FUNCTION_BLOCK FB_DriveInv IMPLEMENTS I_Drive
VAR
	//HMI
	_autoLed			: FB_Led;			//obiekt diody LED stacyjka SCADA - auto
	_supplyLed			: FB_Led;			//obiekt diody LED stacyjka SCADA - zasilanie
	_fwdLed				: FB_Led;			//obiekt diody LED Stacyjka SCADA - kierunek
	_revLed				: FB_LED;			//obiekt diody LED Stacyjka SCADA - kierunek do tyłu
	_stateLed			: FB_LedColorful;	//obiekt etykiety LABEL stacyjka SCADA
	_statusLabel    	: FB_Label;			//obiekt etykiety LABEL sstatus


	// Latch RUN tylko w Drive
    _reqFwd, _reqRev 	: BOOL;
	_fault			 	: BOOL;
	
	// poziomy do styczników
    _cmdFwd, _cmdRev 	: BOOL;
	
	//zezwolenia
	_safetyOk       	: BOOL := TRUE;	// Zawsze TRUE jesli brak przekazników safety
    _permOk	 		 	: BOOL := TRUE;    // „zawsze TRUE”, jeśli brak per-permitu
	
		
	// instancje styczników – referencje wiązane w FB_init
    Fwd					: FB_Contactor( en := _cmdFwd);
    Rev 				: FB_Contactor( en := _cmdRev);
	
	//stan napędu
	_termFuseOk		 	: FB_TermFuse;		//obiekt wylacznika silnikowego fizyczne szafa sterownicza
	_isRunning		 	: BOOL; 
	_isRunningRev 	 	: BOOL;
	
	//czas pracy
	_fbWorkTimeCounter	: FB_WorkTimeCounter; //obiekt do zarzadzania czasem pracy napędu
	_stWorkTime			: ST_WorkTime;		 //struktura przechowywania czasu pracy
	_wtEnable			: BOOL;				//uruchamia licznik czasu pracy
	
	//nastawa i aktualna czestotliwość w HZ pracy
	_rSetHz 			: REAL;   // bufor nastawy (ostatnio zadane)
    _rActHz				: REAL;   // ostatni odczyt z falownika
	
	//struktura rejestrowana do wymiany danych z modbusem
	_stInverter	   		: ST_Inverter; //struktura wymiany danych i ustawień poprzez modbus
	_idx			    : UINT; //numer instancji
		
END_VAR

PROPERTY AtSpeed : BOOL
GET
AtSpeed := EtaHasBit(_stInverter.wInvStatusWord, E_EtaBit.AtSpeed);
END_GET
END_PROPERTY

PROPERTY CommOk : BOOL
GET
CommOk := _stInverter.bCommOk;
END_GET
SET
_stInverter.bCommOk := CommOk;
END_SET
END_PROPERTY

METHOD Cycle : BOOL
// ciało FB (co cykl)

//błąd napedu
_fault := NOT _termFuseOk.IsActive; //zadziałał termik lub falownik ma bład z słowa statusu 

_cmdFwd := _reqFwd AND NOT _reqRev AND _safetyOk AND _permOk AND NOT _fault;
_cmdRev := _reqRev AND NOT _reqFwd AND _safetyOk AND _permOk AND NOT _fault;

//instancje styczników (przekażników) załączajaccyh przód tył
Fwd();  Rev();

//----w przypadku falownika potwierdzamy ze slowa statusu falownika maskuajc odpowiedni bit pobierammmy getterem
_isRunning    := IsRunning;
_isRunningRev := IsRunningRev;

//Odliczanie czasu pracy
_fbWorkTimeCounter.Execute(_wtEnable AND (_isRunning OR _isRunningRev));
_stWorkTime := _fbWorkTimeCounter.WorkTime;


//ustawienia _stInverter tylko przekazujemy Hz, SlaveId, InvType przekazane w FB_INIT 
_stInverter.rFreqSetPoint := _rSetHz;
_rActHz := _stInverter.rFreqActual; //ustaw odczytana actualna czestotliwosc z Modbus

Cycle:=TRUE;
END_METHOD

{warning 'add property implementation'}
PROPERTY Fault : BOOL
GET
Fault := EtaHasBit(_stInverter.wInvStatusWord, E_EtaBit.Fault);
END_GET
END_PROPERTY

METHOD FB_init : BOOL
VAR_INPUT
	bInitRetains : BOOL; // if TRUE, the retain variables are initialized (warm start / cold start)
	bInCopyCode  : BOOL;  // if TRUE, the instance afterwards gets moved into the copy code (online change)
	bDeviceId    : BYTE;           //Adres Slave falownika
	eDeviceType	 : E_InvType; //Enum z typem falownika	
END_VAR

VAR
	fbDriveRegistry : FB_DriveRegistry;

END_VAR
//UStaw adres slava oraz model falownika
THIS^._stInverter.nSlaveId := bDeviceId;
THIS^._stInverter.eInvModel := eDeviceType;


//Rejestracja struktury
fbDriveRegistry.Register( ADR(_stInverter), index => _idx);   // <<< statyczna metoda klasy
END_METHOD

PROPERTY InvStatWord : WORD
GET
InvStatWord := _stInverter.wInvStatusWord;
END_GET
SET
_stInverter.wInvStatusWord	:= InvStatWord;
END_SET
END_PROPERTY

{warning 'add property implementation'}
PROPERTY IsRunning : BOOL
GET
IsRunning := EtaHasBit(_stInverter.wInvStatusWord, E_EtaBit.OperEnabled) AND NOT EtaHasBit(_stInverter.wInvStatusWord, E_EtaBit.DirRev);
END_GET
END_PROPERTY

{warning 'add property implementation'}
PROPERTY IsRunningRev : BOOL
GET
IsRunningRev := EtaHasBit(_stInverter.wInvStatusWord, E_EtaBit.DirRev);
END_GET
END_PROPERTY

{warning 'add method implementation '}
METHOD ResetFault : BOOL
ResetFault := TRUE;
END_METHOD

PROPERTY SetAutoLed : BOOL
GET
SetAutoLed:=_autoLed.State;
END_GET
SET
_autoLed.State:=SetAutoLed;
END_SET
END_PROPERTY

PROPERTY SetFwdLed : BOOL
GET
SetFwdLed := _fwdLed.State;
END_GET
SET
_fwdLed.State := SetFwdLed;
END_SET
END_PROPERTY

PROPERTY SetLedEnum : E_DriveLedState
SET
_stateLed.StateAsEnum := SetLedEnum;
END_SET
END_PROPERTY

PROPERTY SetLedInt : INT
GET
SetLedInt := _stateLed.StateAsInt;
END_GET
END_PROPERTY

PROPERTY SetRevLed : BOOL
GET
END_GET
SET
END_SET
END_PROPERTY

PROPERTY SetStatusLabel : STRING
GET
SetStatusLabel := _statusLabel.Text;
END_GET
SET
_statusLabel.Text := SetStatusLabel;
END_SET
END_PROPERTY

PROPERTY SetSupplyLed : BOOL
GET
SetSupplyLed := _supplyLed.State;
END_GET
SET
_supplyLed.State := SetSupplyLed;
END_SET
END_PROPERTY

METHOD SetWorkCounter : BOOL
VAR_INPUT
	bEnable	:	BOOL;
END_VAR
_wtEnable := bEnable;
END_METHOD

PROPERTY SlaveId : BYTE
GET
SlaveId:=_stInverter.nSlaveId;
END_GET
END_PROPERTY

PROPERTY SpeedAct_Hz : REAL
GET
SpeedAct_Hz := _rActHz;
END_GET
SET
_rActHz := SpeedAct_Hz;
END_SET
END_PROPERTY

PROPERTY SpeedSet_Hz : REAL
GET
SpeedSet_Hz :=_rSetHz;
END_GET
SET
_rSetHz := SpeedSet_Hz;
END_SET
END_PROPERTY

{warning 'add method implementation '}
METHOD StartForward : BOOL
_reqFwd := TRUE;
_reqRev := FALSE;   // antykolizja
StartForward := TRUE;
END_METHOD

{warning 'add method implementation '}
METHOD StartReverse : BOOL
_reqRev := TRUE;
_reqFwd := FALSE;   // antykolizja
StartReverse := TRUE;
END_METHOD

{warning 'add method implementation '}
METHOD Stop : BOOL
_reqFwd := FALSE;
_reqRev := FALSE;
Stop := TRUE;
END_METHOD

PROPERTY TermFuseActive : BOOL
GET
TermFuseActive:=_termFuseOk.IsActive;
END_GET
END_PROPERTY

PROPERTY WorkTime : ST_WorkTime
GET
WorkTime := _stWorkTime;
END_GET
END_PROPERTY

END_FUNCTION_BLOCK

(* stored: Version 1.1.0.1, ProductVersion 3.1.4024.15
   POU FB_DriveInv: Id {998f157d-98f4-4a1d-a525-f21d6db1752c}, SpecialFunc None
   Folder Properties: Id {ab91cccc-fd8c-48aa-9c62-433bf5d3d562}
   Folder HMI: Id {7a1cb371-1287-48fe-8bf1-6e2347960f87}
   Folder Speed: Id {13697b6e-c152-48ca-8364-c7b21cb26641}
   Folder Status: Id {60b0fbd8-c2fb-4a59-b06b-b79a810a4fce}
   Property AtSpeed: Id {7ebf9d48-ac3a-46b6-bd4f-79f980ebea2b}
   Get Get: Id {26deacff-d269-4f49-89d4-88876f43fb3e}
   Property CommOk: Id {09728eaa-9276-4104-b401-530e764e10d2}
   Get Get: Id {ddad8bc1-dd14-45f3-8603-2ba4970767b0}
   Set Set: Id {6b7d97cd-b407-459b-a06c-07a364894300}
   Method Cycle: Id {5ff6d694-42e7-4915-a107-7ec0910a6f23}
   Property Fault: Id {52a188d9-3e41-429e-817b-3f62a2e7e738}
   Get Get: Id {db474149-d812-4fda-97a3-a696d66daf32}
   Method FB_init: Id {ec766e15-c923-48ff-bc8b-53f7a80f7482}
   Property InvStatWord: Id {3c15abbd-5053-434a-a0ba-d8c51ce0164d}
   Get Get: Id {db1818b5-ed42-4a17-95d6-e6ce25aeb156}
   Set Set: Id {76e7d4f2-7cda-41e2-bc52-1673a71231c8}
   Property IsRunning: Id {d62d39a7-703c-4002-aa4a-0ed906638fe8}
   Get Get: Id {ea63fa90-ea31-4184-bbe4-465e0e3fa95c}
   Property IsRunningRev: Id {e2de8772-48bb-471a-a81b-910da806c580}
   Get Get: Id {36949d3e-2d2d-462a-b0fb-0d3c957fe3a5}
   Method ResetFault: Id {15dd322f-e0ee-4399-a95c-70372cb8d9be}
   Property SetAutoLed: Id {bcb83271-1cf3-43ea-9f19-44a9280bb696}
   Get Get: Id {f1762002-d8fc-4f3e-8dd8-1079f692b77a}
   Set Set: Id {f2c95e51-7214-460c-853c-e3f5c007ecf2}
   Property SetFwdLed: Id {131869f1-e68b-4c6c-b4f8-dac85d1233be}
   Get Get: Id {0fb773dd-b98d-481b-9bf5-1e4021df1234}
   Set Set: Id {22d80d52-6c39-4562-b222-90b76ff6a526}
   Property SetLedEnum: Id {a418d578-11da-48f4-862f-892a41df79e4}
   Set Set: Id {adf10085-ec57-4ee2-8d39-c544ba2f42cf}
   Property SetLedInt: Id {c94d2d0c-c416-4c9c-825f-af6f07095bb7}
   Get Get: Id {bd38b4bb-648d-4ac4-881b-b1cf76137d6a}
   Property SetRevLed: Id {9b8a98f5-39dc-41af-83d5-8ae024318d20}
   Get Get: Id {5b8ecbe8-ce35-4b92-9e0f-e469cbfdc363}
   Set Set: Id {4b1e470a-4ca3-4cc2-b066-50ec00d1f3b6}
   Property SetStatusLabel: Id {e2bbff0a-60f7-410c-b1ab-103abb8901fd}
   Get Get: Id {2778f0b1-a9fd-49cb-8c1a-ecdbf2c8001e}
   Set Set: Id {563390b6-6d0e-4128-af15-f368a16aaa2a}
   Property SetSupplyLed: Id {3200588f-4438-4463-891b-78da2541a960}
   Get Get: Id {ad1abc8e-5445-4808-8540-43632081bec9}
   Set Set: Id {e29dd435-b94b-4139-b86b-0fae42cb2d2c}
   Method SetWorkCounter: Id {18f101cd-d9a2-48ed-b60d-6b15cc8fc25e}
   Property SlaveId: Id {e4c3367f-856e-403a-ad42-306a7994fec4}
   Get Get: Id {320b3815-6d26-467d-b2a4-d543f1bffff2}
   Property SpeedAct_Hz: Id {e897d20c-aba5-41a8-975b-c4c3ffe72dbb}
   Get Get: Id {b54eb1f0-5bc6-411e-9840-9dccc96e7315}
   Set Set: Id {3ef0ab9e-53e0-41b0-8785-6000730ff14b}
   Property SpeedSet_Hz: Id {f274a3c5-d2bb-4899-bf76-292d814a9783}
   Get Get: Id {a98f2280-3112-4649-8dd2-6379c026f46d}
   Set Set: Id {cbda811c-60d8-4250-864e-3dd793356939}
   Method StartForward: Id {003d36e1-d318-48ec-af4b-d479e535378b}
   Method StartReverse: Id {0ea47be1-b422-400c-ae22-25031beeffc7}
   Method Stop: Id {b75b28f3-0cd6-48ad-bf32-26bf81ddd6ce}
   Property TermFuseActive: Id {9cfc7bb2-0739-44d5-b63d-a90e1b63f8e1}
   Get Get: Id {a3f039ae-4077-4afb-b068-cccaf089f702}
   Property WorkTime: Id {cf99b721-49e6-4878-b917-5a7debef1ed3}
   Get Get: Id {ce67d592-f44b-4931-b88b-2c6c1dfe6336} *)
